{attribute addProperty BoxType "KL8001-0002"}
{attribute addProperty Id "Channel_1Channel_1D3D9A8600"}
{attribute addProperty CRC "3259744062"}
{attribute addProperty SizeInBites "0"}
{attribute addProperty SizeInBytes "0"}
TYPE KL_C24BBF3E :
STRUCT
	{attribute addProperty Name "Channel_1"}
	Channel_1 : Channel_1D3D9A86;
END_STRUCT
END_TYPE

(* stored: Version 1.2.0.0, ProductVersion 3.1.4024.9
   DUT KL_C24BBF3E: Id {98e8f9c3-6491-499f-a2ce-aa4f4d8762fb} *)
